PROGRAM OP130_RH_Initialization_Seq
VAR
END_VAR





CASE OP130_RH_Homing_Seq OF 
	
       	0: IF (OP130_Auto AND NOT OP130_HomeRunning AND  NOT OP130_ErrorActive AND  NOT OP130_AutoRunning AND NOT OP130_StepRunning	 AND NOT OP130_Temp_Home_OK) THEN
       		  OP130_HomeRunning:=TRUE;
       		  OP130_RH_Homing_Seq:=10;	
       	   END_IF
	   
	    10:IF SR130_stManualModeAxis_RH_Vert_Servo.actualPosition >=61  THEN
		      OP130_RH_Homing_Seq:=20;
	        ELSE
		      OP130_RH_Homing_Seq:=90;
		    END_IF
	   
	   20: IF (OP130_HomeRunning AND OP130_HMI_Homing)THEN 
		     // OP130_GVL.SR130_RH_Vert_Servo.fTargetPosition:=SR130_HMI_Servo_CylWork_Position;
		    // OP130_GVL.SR130_RH_Vert_Servo.fTargetVelocity:=SR130_HMI_Servo_CylWork_Velocity;
		      SR130_RH_Servo_Control.Position:=SR130_HMI_Servo_CylWork_Position;
			  SR130_RH_Servo_Control.Velocity:=SR130_HMI_Servo_CylWork_Velocity;
		      OP130_RH_Homing_Seq:=30;
	       END_IF
	   
	   30: IF (OP130_HomeRunning AND OP130_HMI_Homing)THEN 
		   //  SR130_RH_Abs_Move_Start:=TRUE;
			 SR130_RH_Servo_Control.ABSmove_Start:=TRUE;
			 OP130_RH_Homing_Seq:=40;
	       END_IF
		   
	   40:IF (OP130_HomeRunning AND OP130_HMI_Homing)THEN 
		     IF OP130_GVL.SR130_RH_Servo_Control.Axis_In_Pos THEN
			// SR130_RH_Abs_Move_Start:=FALSE;
			    SR130_RH_Servo_Control.ABSmove_Start:=FALSE;
			    OP130_RH_Homing_Seq:=50;
		     END_IF
	      END_IF
		  
	   50:IF (OP130_HomeRunning AND OP130_HMI_Homing)THEN 
		   IF CR130_RH_Rot_Cyl.Position2 THEN
			   OP130_RH_Homing_Seq:=60; 
		    ELSE
		      OP130_GVL.CR130_RH_Rot_Cyl.HomingCmd2:= TRUE;
		      OP130_GVL.CR130_RH_Rot_Cyl.HomingCmd1:= FALSE;
	       END_IF
	   END_IF
	   
	   60:IF (OP130_HomeRunning AND OP130_HMI_Homing)THEN 
		    //OP130_GVL.SR130_RH_Vert_Servo.fTargetPosition:=SR130_HMI_Servo_Rotation_Position;
		    //OP130_GVL.SR130_RH_Vert_Servo.fTargetVelocity:=SR130_HMI_Servo_Rotation_Velocity;
		     SR130_RH_Servo_Control.Position:=SR130_HMI_Servo_Rotation_Position;
		     SR130_RH_Servo_Control.Velocity:=SR130_HMI_Servo_Rotation_Velocity;
		     OP130_RH_Homing_Seq:=70;
	      END_IF
	   
	   70: IF (OP130_HomeRunning AND OP130_HMI_Homing)THEN 
		     //SR130_RH_Abs_Move_Start:=TRUE;
			   SR130_RH_Servo_Control.ABSmove_Start:=TRUE;
			   IF  OP130_GVL.SR130_RH_Servo_Control.Axis_In_Pos THEN
				 // SR130_RH_Abs_Move_Start:=FALSE;
				  SR130_RH_Servo_Control.ABSmove_Start:=FALSE;
				  OP130_RH_Homing_Seq:=80;
			   END_IF
	       END_IF
		   
	80:IF (OP130_HomeRunning AND OP130_HMI_Homing)THEN 
		  IF OP130_GVL.CR130_RH_Rot_Cyl.Position1 THEN
			OP130_RH_Homing_Seq:=90;
		  ELSE
				OP130_GVL.CR130_RH_Rot_Cyl.HomingCmd1:= TRUE;
				OP130_GVL.CR130_RH_Rot_Cyl.HomingCmd2:= FALSE;
		  END_IF
	   END_IF
	
	90:IF (OP130_HomeRunning AND OP130_HMI_Homing)THEN  
		//  OP130_GVL.SR130_RH_Vert_Servo.fTargetPosition:=0.0;
		//  OP130_GVL.SR130_RH_Vert_Servo.fTargetVelocity:=10;
		  SR130_RH_Servo_Control.Position :=0.0;
		  SR130_RH_Servo_Control.Velocity :=10;
		  OP130_RH_Homing_Seq:=100;
	   END_IF
	
	100:IF (OP130_HomeRunning AND OP130_HMI_Homing)THEN 
           SR130_RH_Abs_Move_Start:=TRUE;
	       SR130_RH_Servo_Control.ABSmove_Start:=TRUE;
			IF SR130_RH_Servo_Control.Axis_In_Pos THEN
			//   SR130_RH_Abs_Move_Start:=FALSE;
			   SR130_RH_Servo_Control.ABSmove_Start:=FALSE;
			   OP130_RH_Homing_Seq:=110;
			END_IF
		END_IF
		
	110: 
		OP130_HomeRunning:=FALSE;
		OP130_RH_Homing_Seq:=0;
	
END_CASE

END_PROGRAM

(* stored: Version 1.1.0.1, ProductVersion 3.1.4024.11
   POU OP130_RH_Initialization_Seq: Id {0590351b-9308-461f-98bc-e3f7869fe039}, SpecialFunc None *)
